# EPICS autosave request: iocBoot/iocUSB1208/auto_settings.req
file "USB1208_settings.req", P=$(P)
